(* PLC project Scenario0_Final.project, CODESYS CODESYS V3.5 SP4 Patch 4 *)
(* stored: creationDateTime 2014-06-25T14:55:42.4423777, modificationDateTime 2014-06-20T17:27:16 *)

FUNCTION_BLOCK Magazin
  VAR_INPUT
    SliderNotMovedOut : BOOL;
    SliderMovedOut : BOOL;
    WorkpieceReady : BOOL;
    CraneDown : BOOL;
    CraneUp : BOOL;
    CraneOnConveyor : BOOL;
    CraneOnMagazin : BOOL;
    CraneSucked : BOOL;
    StartButtonMagazin : BOOL;
    SFCReset : BOOL;
    StartVar : BOOL;
  END_VAR
  VAR_OUTPUT
    MagazinSlider : BOOL;
    MagazinGreenLamp : BOOL;
    StartCommandMagazin : BOOL;
  END_VAR
  VAR
    interconnectMagazineStartCommand : BOOL;
    SFCInit : BOOL;
  END_VAR

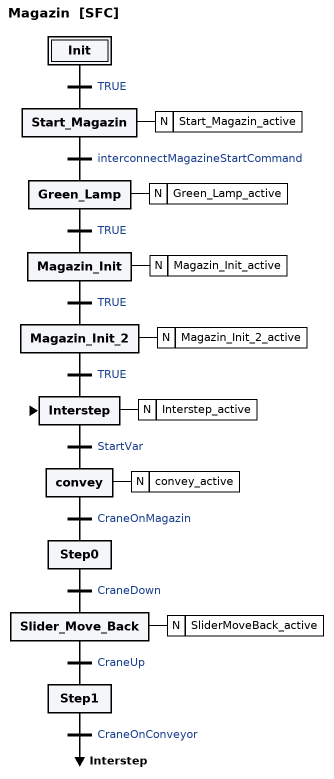
INITIAL_STEP Init:
END_STEP
TRANSITION FROM Init TO Start_Magazin
  := TRUE;
END_TRANSITION
STEP Start_Magazin:
  Start_Magazin_active(N);
END_STEP
TRANSITION FROM Start_Magazin TO Green_Lamp
  := interconnectMagazineStartCommand;
END_TRANSITION
STEP Green_Lamp:
  Green_Lamp_active(N);
END_STEP
TRANSITION FROM Green_Lamp TO Magazin_Init
  := TRUE;
END_TRANSITION
STEP Magazin_Init:
  Magazin_Init_active(N);
END_STEP
TRANSITION FROM Magazin_Init TO Magazin_Init_2
  := TRUE;
END_TRANSITION
STEP Magazin_Init_2:
  Magazin_Init_2_active(N);
END_STEP
TRANSITION FROM Magazin_Init_2 TO Interstep
  := TRUE;
END_TRANSITION
STEP Interstep:
  Interstep_active(N);
END_STEP
TRANSITION FROM Interstep TO convey
  := StartVar;
END_TRANSITION
STEP convey:
  convey_active(N);
END_STEP
TRANSITION FROM convey TO Step0
  := CraneOnMagazin;
END_TRANSITION
STEP Step0:
END_STEP
TRANSITION FROM Step0 TO Slider_Move_Back
  := CraneDown;
END_TRANSITION
STEP Slider_Move_Back:
  SliderMoveBack_active(N);
END_STEP
TRANSITION FROM Slider_Move_Back TO Step1
  := CraneUp;
END_TRANSITION
STEP Step1:
END_STEP
TRANSITION FROM Step1 TO Interstep
  := CraneOnConveyor;
END_TRANSITION

ACTION Green_Lamp_active:
                                MagazinGreenLamp := TRUE;
                                    interconnectMagazineStartCommand := FALSE;
                                
                            
END_ACTION

ACTION Magazin_Init_2_active:
                                MagazinSlider := FALSE;
                            
END_ACTION

ACTION SliderMoveBack_active:
                                IF((SliderMovedOut =
                                    TRUE)AND(SliderNotMovedOut = FALSE))THEN
                                    MagazinSlider := FALSE;
                                    END_IF
                                
                            
END_ACTION

ACTION convey_active:
                                IF(SliderNotMovedOut)THEN
                                    MagazinSlider := TRUE;
                                    END_IF
                                
                            
END_ACTION

ACTION Start_Magazin_active:
                                MagazinSlider := FALSE;
                                    MagazinGreenLamp := FALSE;
                                    StartVar := FALSE;
                                    StartCommandMagazin := FALSE;


                                    IF(StartButtonMagazin = TRUE) THEN
                                    interconnectMagazineStartCommand := TRUE;
                                    END_IF
                                
                            
END_ACTION

ACTION Magazin_Init_active:
                                MagazinSlider := TRUE;
                            
END_ACTION

ACTION Interstep_active:
                                StartCommandMagazin := TRUE;
                            
END_ACTION
END_FUNCTION_BLOCK

FUNCTION_BLOCK Crane
  VAR_INPUT
    SliderNotMovedOut : BOOL;
    SliderMovedOut : BOOL;
    WorkpieceReady : BOOL;
    CraneDown : BOOL;
    CraneUp : BOOL;
    CraneOnConveyor : BOOL;
    CraneOnMagazin : BOOL;
    CraneSucked : BOOL;
    StartButtonMagazin : BOOL;
    SFCReset : BOOL;
    StartVar : BOOL;
  END_VAR
  VAR_OUTPUT
    CraneLower : BOOL;
    MagazinVacuumOff : BOOL;
    MagazinVacuumOn : BOOL;
    CraneTurnCounterclockwise : BOOL;
    CraneTurnClockwise : BOOL;
    StartCommandCrane : BOOL;
  END_VAR
  VAR
    interconnectCraneStartCommand : BOOL;
    TimeDelay_Timer : TON;
    TimeDelay_Timer_Duration : TIME := TIME#50ms;
    TimeDelay_Timer_interconnect : BOOL;
    SFCInit : BOOL;
  END_VAR

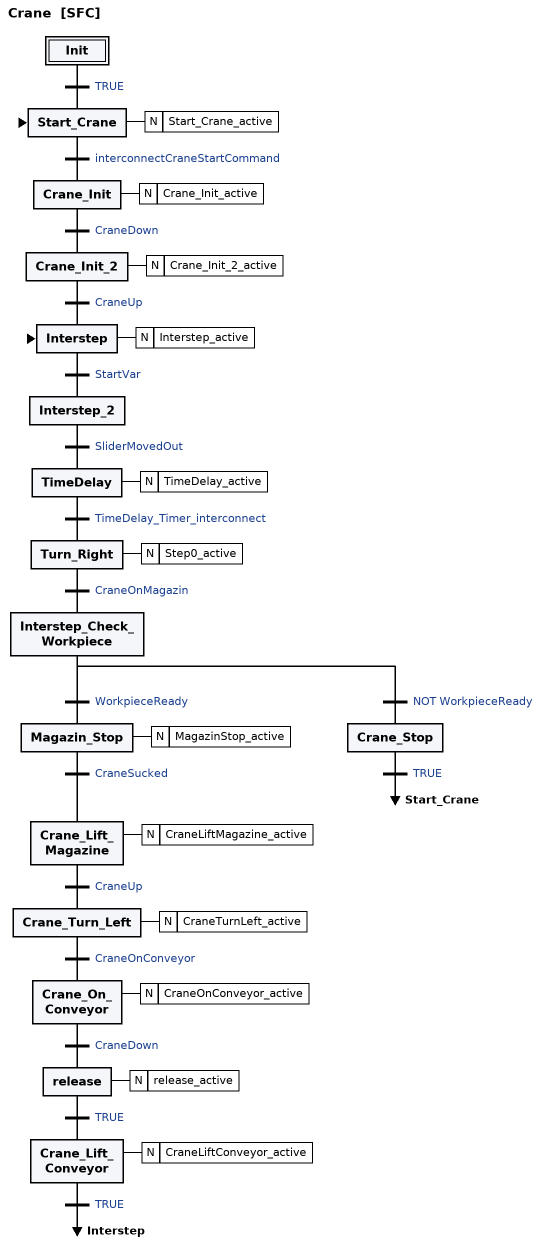
INITIAL_STEP Init:
END_STEP
TRANSITION FROM Init TO Start_Crane
  := TRUE;
END_TRANSITION
STEP Start_Crane:
  Start_Crane_active(N);
END_STEP
TRANSITION FROM Start_Crane TO Crane_Init
  := interconnectCraneStartCommand;
END_TRANSITION
STEP Crane_Init:
  Crane_Init_active(N);
END_STEP
TRANSITION FROM Crane_Init TO Crane_Init_2
  := CraneDown;
END_TRANSITION
STEP Crane_Init_2:
  Crane_Init_2_active(N);
END_STEP
TRANSITION FROM Crane_Init_2 TO Interstep
  := CraneUp;
END_TRANSITION
STEP Interstep:
  Interstep_active(N);
END_STEP
TRANSITION FROM Interstep TO Interstep_2
  := StartVar;
END_TRANSITION
STEP Interstep_2:
END_STEP
TRANSITION FROM Interstep_2 TO TimeDelay
  := SliderMovedOut;
END_TRANSITION
STEP TimeDelay:
  TimeDelay_active(N);
END_STEP
TRANSITION FROM TimeDelay TO Turn_Right
  := TimeDelay_Timer_interconnect;
END_TRANSITION
STEP Turn_Right:
  Step0_active(N);
END_STEP
TRANSITION FROM Turn_Right TO Interstep_Check_Workpiece
  := CraneOnMagazin;
END_TRANSITION
STEP Interstep_Check_Workpiece:
END_STEP
TRANSITION FROM Interstep_Check_Workpiece TO Magazin_Stop
  := WorkpieceReady;
END_TRANSITION
TRANSITION FROM Interstep_Check_Workpiece TO Crane_Stop
  := NOT WorkpieceReady;
END_TRANSITION
STEP Magazin_Stop:
  MagazinStop_active(N);
END_STEP
TRANSITION FROM Magazin_Stop TO Crane_Lift_Magazine
  := CraneSucked;
END_TRANSITION
STEP Crane_Lift_Magazine:
  CraneLiftMagazine_active(N);
END_STEP
TRANSITION FROM Crane_Lift_Magazine TO Crane_Turn_Left
  := CraneUp;
END_TRANSITION
STEP Crane_Turn_Left:
  CraneTurnLeft_active(N);
END_STEP
TRANSITION FROM Crane_Turn_Left TO Crane_On_Conveyor
  := CraneOnConveyor;
END_TRANSITION
STEP Crane_On_Conveyor:
  CraneOnConveyor_active(N);
END_STEP
TRANSITION FROM Crane_On_Conveyor TO release
  := CraneDown;
END_TRANSITION
STEP release:
  release_active(N);
END_STEP
TRANSITION FROM release TO Crane_Lift_Conveyor
  := TRUE;
END_TRANSITION
STEP Crane_Lift_Conveyor:
  CraneLiftConveyor_active(N);
END_STEP
TRANSITION FROM Crane_Lift_Conveyor TO Interstep
  := TRUE;
END_TRANSITION
STEP Crane_Stop:
END_STEP
TRANSITION FROM Crane_Stop TO Start_Crane
  := TRUE;
END_TRANSITION

ACTION CraneTurnLeft_active:
                                CraneTurnCounterclockwise := TRUE;
                                    CraneTurnClockwise := FALSE;
                                
                            
END_ACTION

ACTION Step0_active:
                                CraneTurnClockwise := TRUE;
                                    CraneTurnCounterclockwise := FALSE;
                                
                            
END_ACTION

ACTION CraneOnConveyor_active:
                                CraneTurnCounterclockwise := FALSE;
                                    CraneTurnClockwise := FALSE;
                                    CraneLower := TRUE;
                                
                            
END_ACTION

ACTION MagazinStop_active:
                                CraneTurnClockwise := FALSE;
                                    CraneTurnCounterClockwise := FALSE;
                                    MagazinVacuumOn := TRUE;
                                    MagazinVacuumOff := FALSE;
                                    CraneLower := TRUE;
                                
                            
END_ACTION

ACTION Crane_Init_2_active:
                                CraneLower := FALSE;
                            
END_ACTION

ACTION Start_Crane_active:
                                CraneLower := FALSE;
                                    MagazinVacuumOff := TRUE;
                                    MagazinVacuumOn := FALSE;
                                    CraneTurnCounterclockwise := FALSE;
                                    CraneTurnClockwise := FALSE;;
                                    StartVar := FALSE;
                                    StartCommandCrane := FALSE;


                                    IF(StartButtonMagazin = TRUE) THEN
                                    interconnectCraneStartCommand := TRUE;
                                    END_IF
                                
                            
END_ACTION

ACTION CraneLiftMagazine_active:
                                CraneLower := FALSE;
                            
END_ACTION

ACTION Interstep_active:
                                StartCommandCrane := TRUE;
                            
END_ACTION

ACTION release_active:
                                MagazinVacuumOff := TRUE;
                                    MagazinVacuumOn := FALSE;
                                
                            
END_ACTION

ACTION Crane_Init_active:
                                CraneLower := TRUE;
                                    interconnectCraneStartCommand := FALSE;
                                
                            
END_ACTION

ACTION TimeDelay_active:
                                TimeDelay_Timer(IN:=TRUE,
                                    PT:=TimeDelay_Timer_Duration);
                                    TimeDelay_Timer_interconnect := TimeDelay_Timer.Q;
                                
                            
END_ACTION

ACTION CraneLiftConveyor_active:
                                CraneLower := FALSE;
                            
END_ACTION
END_FUNCTION_BLOCK

PROGRAM Main
  VAR
    Sensor_StartButtonMagazin : BOOL;
    Sensor_MagazinEmergencyStop : BOOL;
    Sensor_MagazinSwitchManuellAutomatic : BOOL;
    Sensor_CraneSucked : BOOL;
    Sensor_CraneDown : BOOL;
    Sensor_CraneUp : BOOL;
    Sensor_SliderNotMovedOut : BOOL;
    Sensor_SliderMovedOut : BOOL;
    Sensor_CraneOnConveyor : BOOL;
    Sensor_CraneOnMagazin : BOOL;
    Sensor_WorkpieceReady : BOOL;
    Sensor_CranePosition : BOOL;
    Actuator_MagazinSlider : BOOL;
    Actuator_CraneLower : BOOL;
    Actuator_MagazinVacuumOn : BOOL;
    Actuator_MagazinVacuumOff : BOOL;
    Actuator_MagazinGreenLamp : BOOL;
    Actuator_MagazinWhiteLamp : BOOL;
    Actuator_CraneTurnCounterclockwise : BOOL;
    Actuator_CraneTurnClockwise : BOOL;
    Mag : Magazin;
    Crane : Crane;
  END_VAR

                        Mag.SliderNotMovedOut := Sensor_SliderNotMovedOut;
                            Mag.SliderMovedOut := Sensor_SliderMovedOut;
                            Mag.CraneOnMagazin := Sensor_CraneOnMagazin;
                            Mag.CraneDown := Sensor_CraneDown;
                            Mag.CraneUp := Sensor_CraneUp;
                            Mag.CraneOnConveyor := Sensor_CraneOnConveyor;
                            Mag.WorkpieceReady := Sensor_WorkpieceReady;
                            Mag.StartButtonMagazin := Sensor_StartButtonMagazin;

                            Actuator_MagazinSlider := Mag.MagazinSlider;
                            Actuator_MagazinGreenLamp := Mag.MagazinGreenLamp;


                            Crane.WorkpieceReady := Sensor_WorkpieceReady;
                            Crane.CraneUp := Sensor_CraneUp;
                            Crane.CraneOnConveyor := Sensor_CraneOnConveyor;
                            Crane.CraneDown := Sensor_CraneDown;
                            Crane.CraneSucked := Sensor_CraneSucked;
                            Crane.CraneOnMagazin := Sensor_CraneOnMagazin;
                            Crane.SliderMovedOut := Sensor_SliderMovedOut;
                            Crane.StartButtonMagazin := Sensor_StartButtonMagazin;

                            Actuator_CraneTurnCounterclockwise := Crane.CraneTurnCounterclockwise;
                            Actuator_CraneTurnClockwise := Crane.CraneTurnClockwise;
                            Actuator_CraneLower := Crane.CraneLower;
                            Actuator_MagazinVacuumOff := Crane.MagazinVacuumOff;
                            Actuator_MagazinVacuumOn := Crane.MagazinVacuumOn;


                            IF((Sensor_MagazinEmergencyStop))THEN
                            Mag();
                            Crane();
                            IF((Actuator_MagazinGreenLamp))THEN
                            IF((Crane.StartCommandCrane) AND (Mag.StartCommandMagazin))THEN
                            Crane.StartVar := TRUE;
                            Mag.StartVar := TRUE;
                            END_IF
                            END_IF
                            Crane.SFCReset := FALSE;
                            Mag.SFCReset := FALSE;
                            ELSIF ((NOT Sensor_MagazinEmergencyStop))THEN
                            Actuator_MagazinSlider := FALSE;
                            Actuator_CraneLower := FALSE;
                            Actuator_MagazinVacuumOn := FALSE;
                            Actuator_MagazinVacuumOff := TRUE;
                            Actuator_MagazinGreenLamp := FALSE;
                            Actuator_CraneTurnCounterclockwise := FALSE;
                            Actuator_CraneTurnClockwise := FALSE;

                            Crane.SFCReset := TRUE;
                            Mag.SFCReset := TRUE;

                            Crane.StartVar := FALSE;
                            Mag.StartVar := FALSE;
                            END_IF
                        
                    
END_PROGRAM
